FUNCTION_BLOCK AutoMove
VAR_INPUT
END_VAR
VAR_OUTPUT
END_VAR
VAR
END_VAR

IF AUTO.Status > 0 AND AUTO.Status < AUTO.N THEN
	IF AUTO.Current.A <> AUTO.Komande0[AUTO.Status].A  THEN
		AUTO.MotorIzbira := 1;
		IF AUTO.Current.A > AUTO.Komande0[AUTO.Status].A THEN
			AUTO.VrtenjeSmer := TRUE;
		ELSE
			AUTO.VrtenjeSmer := FALSE;
		END_IF
		AUTO.VrtenjePremik := TRUE;
	ELSIF AUTO.Current.Y <> AUTO.Komande0[AUTO.Status].Y  THEN
		AUTO.MotorIzbira := 3;
		IF AUTO.Current.Y > AUTO.Komande0[AUTO.Status].Y THEN
			AUTO.IztegSmer := TRUE;
		ELSE
			AUTO.IztegSmer := FALSE;
		END_IF
		AUTO.IztegPremik := TRUE;
	ELSIF AUTO.Current.Z <> AUTO.Komande0[AUTO.Status].Z  THEN
		AUTO.MotorIzbira := 2;
		IF AUTO.Current.Z > AUTO.Komande0[AUTO.Status].Z THEN
			AUTO.DvigSmer := TRUE;
		ELSE
			AUTO.DvigSmer := FALSE;
		END_IF
		AUTO.DvigPremik := TRUE;
	ELSIF AUTO.Current.P <> AUTO.Komande0[AUTO.Status].P  THEN
		AUTO.MotorIzbira := 4;
		IF AUTO.Current.P > AUTO.Komande0[AUTO.Status].P THEN
			AUTO.PrijemSmer := TRUE;
		ELSE
			AUTO.PrijemSmer := FALSE;
		END_IF
		AUTO.PrijemPremik := TRUE;
	ELSE
		AUTO.VrtenjePremik := FALSE;
		AUTO.DvigPremik := FALSE;
		AUTO.IztegPremik := FALSE;
		AUTO.PrijemPremik := FALSE;
		AUTO.Status := AUTO.Status + 1;
	END_IF
END_IF

END_FUNCTION_BLOCK

(* stored: Version 1.1.0.1, ProductVersion 3.1.4024.12
   POU AutoMove: Id {f87ec304-afbe-4cdb-bf11-12928f5bbd8d}, SpecialFunc None *)
